Staubli VAL3: FibraHSI.dtx

public frame fFrame = {x=317.444674, y=77.778782, z=-312.57185, rx=-0.864374, ry=0.359034, rz=1.064618, fatherId=world[0]}
public jointRx jJointRx = {j1=45, j2=45, j3=45, j4=45, j5=45, j6=45}
public jointRx jJointRxZeros
public mdesc mMdescFibra = {accel=5, vel=10, decel=5, tmax=10, rmax=10, leave=10, reach=10, blend=cartesian}
public mdesc mMdescMov = {accel=90, decel=90, tmax=99.999, rmax=99.999, blend=cartesian}
mdesc mNomSpeed
num nNumPort = 1000
num nReceiveByte[64]
num nResult
num nXPosButTxt[9]
  [2] = 5
  [3] = 10
  [4] = 15
  [5] = 20
  [6] = 25
  [7] = 30
  [8] = 35
num nYPosButTxt = 13
pointRx pPointRxOrigin = {ry=180, fatherId=fFrame[0]}
pointRx pTempSocket = {fatherId=fFrame[0]}
public sio sSio = {link=Socket\fibra_ser}
public string sInputMsg
public string sOutputMsg
tool ftool = {x=76.72, y=-0.63, z=152.93, fatherId=flange[0], ioLink=valve1}
public tool tTool = {z=20, fatherId=flange[0], ioLink=valve1}
string sOutputMsgLog
